PROGRAM MAIN
VAR		
	//INPUTS
	PrePump_Pressure_Int AT %I* : INT;
	Chamber_Penning_Int  AT %I* : INT;
	Chamber_Pirani_Int   AT %I* : INT;	
	GasLine_Pirani_Int   AT %I* : INT;
	Sample_BodyTemp      AT %I* : INT;					// Oven temperatures in 0.01 degC
	Sample_CapTemp       AT %I* : INT;
	Sample_TipTemp       AT %I* : INT;	
	Magnet_Temp          AT %I* : INT;
	
	Flow_Valve 			 AT %I* : INT;                  // Gas flow valve conductance 0-10 V
	
	TurboTOF_NO AT %I* : BOOL;	
	TurboTOF_ERR AT %I* : BOOL;
		
	
	// IMPORTANT! 
	// LEYBOLD AND BECKHOOF PLC USE DIFFERENT BYTE ORDER, be careful when linking to profibus
	// LEYBOLD:   0  1  2  3  4  5  6  7  8  9  10 11 12 13 14 15
	// BECKHOFF:  8  9  10 11 12 13 14 15 0  1  2  3  4  5  6  7 
	TurboMain_Overtemp AT %I* : BOOL;
	TurboMain_NO AT %I* : BOOL;
	TurboMain_ERR AT %I* : BOOL;
	TurboMain_Freq AT %I* : UINT;
	
	//OUTPUTS
	Penning_Enable AT %Q* : BOOL;
	LVPS_ON AT %Q* : BOOL;
	MPreVac_Valve AT %Q*: BOOL;
	TOFPreVac_Valve AT %Q* : BOOL;

	TurboTOF_enable AT %Q* : BOOL;
	TurboMain_enable AT %Q*: BOOL;
	TurboMain_Control AT %Q* : BOOL;

	Flow_Valve_Set AT %Q* : INT;    // Flow valve setpoint
	
	FlashInterlock AT %Q* : BOOL;	
	HVPS_ON AT %Q* : INT;
	Lamp1_Enable AT %Q* : BOOL;
	
	//ADS inputs: CONTROL PARAMETERS (PLC reads values and acts accordignly, ADS clients should set these values)
	GasLine_Enable :    BOOL := FALSE;
	Pumps_Enable :      BOOL := FALSE;      // Start pumping sequence
	PreVac_Valve_Lock : BOOL := FALSE;		// Ovverides auto valves and close prevac valves
	
	Sample_Flow_Set : REAL := 0;
	
	SampleX_MotionEnable : BOOL := FALSE;     // Motion enables and setpoints input
	SampleY_MotionEnable : BOOL := FALSE;  	
	SampleZ_MotionEnable : BOOL := FALSE;  	
	SampleX_MotionStop    : BOOL := FALSE;
	SampleY_MotionStop    : BOOL := FALSE;
	SampleZ_MotionStop    : BOOL := FALSE;
	
	FrameX_MotionEnable  : BOOL := FALSE;
	FrameY_MotionEnable  : BOOL := FALSE;
	FrameX_MotionStop     : BOOL := FALSE;
	FrameY_MotionStop     : BOOL := FALSE;
	
	MagnetY_MotionEnable : BOOL := FALSE;
	MagnetY_MotionStop    : BOOL := FALSE;
	
	SampleX_SetPoint : REAL := 0;
	SampleY_SetPoint : REAL := 0;
	SampleZ_SetPoint : REAL := 0;
	FrameX_SetPoint  : REAL := 0;
	FrameY_SetPoint  : REAL := 0;
	MagnetY_SetPoint  : REAL := 0;
	
	//ADS outputs: READ ONLY (PLC updates them at every cycle, ADS clients should just read)
	Chamber_Pressure : REAL;				// Main chamber pressure in mBars
	GasLine_Pressure : REAL;
	PreVac_Pressure  : REAL;                // PrePump line pressure
	PreVacValves_Open: BOOL;	            // Are valves open?

	Sample_Flow : REAL;
	
	TurboPump_ON: BOOL;
	TurboError: BOOL;	
	Turbo_NO:    BOOL;
	
	//Other vars
	PreVac_OK :  BOOL;						// Good prevacuum 
	MainVac_OK : BOOL;
	MainVac_TurboOK : BOOL;
	Oven_OverTEMP: BOOL;
	Pressure_Chamber_Manager: PressureChamber_MNG;
	
	//MOTION 
	manageAx_SampleX: manageAxis;
	manageAx_SampleY: manageAxis;
	manageAx_SampleZ: manageAxis;
	manageAx_FrameX: manageAxis;
	manageAx_FrameY: manageAxis;
	manageAx_MagnetY: manageAxis;	
		
	FrameX : AXIS_REF;
	FrameY : AXIS_REF;
	SampleZ : AXIS_REF;
	SampleX : AXIS_REF;
	SampleY : AXIS_REF;
	MagnetY : AXIS_REF;
	
	SampleX_Fw_End AT %I* : BOOL; // Limit switches
	SampleX_Bw_End AT %I* : BOOL;
	SampleY_Fw_End AT %I* : BOOL;
	SampleY_Bw_End AT %I* : BOOL; 
	SampleZ_Fw_End AT %I* : BOOL;
	SampleZ_Bw_End AT %I* : BOOL;  
	
	FrameX_Fw_End AT %I* : BOOL;
	FrameX_Bw_End AT %I* : BOOL; 
	FrameY_Fw_End AT %I* : BOOL;
	FrameY_Bw_End AT %I* : BOOL; 
	
	MagnetY_Fw_End AT %I* : BOOL;
	MagnetY_Bw_End AT %I* : BOOL;
END_VAR

//*** PROCESS INPUTS ***
//Get pressures in mbar (from ADC value)
Pressure_Chamber_Manager(penningInt := Chamber_Penning_Int, piraniInt := Chamber_Pirani_Int, penningOn => Penning_enable, pressureOut => Chamber_Pressure);
PreVac_Pressure := ConvertPressure_Pirani(PrePump_Pressure_Int);
GasLine_Pressure := ConvertPressure_Pirani(GasLine_Pirani_Int);

//*** MOTION ***
//Move axes
manageAx_SampleX(axis := SampleX, setPoint := SampleX_SetPoint, speed := PARAM.Sample_Movement_Speed, 
		 enable := SampleX_MotionEnable, stop:= SampleX_MotionStop, fwLimit := SampleX_Fw_End, bwLimit := SampleX_Bw_End);
		 
manageAx_SampleY(axis := SampleY, setPoint := SampleY_SetPoint, speed := PARAM.Sample_Movement_Speed, 
		 enable := SampleY_MotionEnable, stop:= SampleY_MotionStop, fwLimit := SampleY_Fw_End, bwLimit := SampleY_Bw_End);	 

manageAx_SampleZ(axis := SampleZ, setPoint := SampleZ_SetPoint, speed := PARAM.Sample_Movement_Speed, 
		 enable := SampleZ_MotionEnable, stop:= SampleZ_MotionStop, fwLimit := SampleZ_Fw_End, bwLimit := SampleZ_Bw_End);
		 
manageAx_FrameX(axis := FrameX,  setPoint := FrameX_SetPoint,  speed := PARAM.Frame_Movement_Speed , 
		 enable := FrameX_MotionEnable, stop:= FrameX_MotionStop, fwLimit := FrameX_Fw_End,  bwLimit := FrameX_Bw_End);

manageAx_FrameY(axis := FrameY,  setPoint := FrameY_SetPoint,  speed := PARAM.Frame_Movement_Speed , 
		 enable := FrameY_MotionEnable, stop:= FrameY_MotionStop, fwLimit := FrameY_Fw_End,  bwLimit := FrameY_Bw_End);
		 
manageAx_MagnetY(axis := MagnetY, setPoint := MagnetY_SetPoint, speed := PARAM.Sample_Movement_Speed, 
		 enable := MagnetY_MotionEnable, stop:= MagnetY_MotionStop, fwLimit := MagnetY_Fw_End, bwLimit := MagnetY_Bw_End);
		 
		 
//*** SAFETY CHECKS ***
// Compute status variables
Oven_OverTEMP   := Sample_BodyTemp > PARAM.Oven_MaxTemp OR Sample_TipTemp > PARAM.Oven_MaxTemp; // OR Sample_CapTemp > PARAM.Oven_MaxTemp Prevent overtemp of oven
TurboError 		:= TurboTOF_ERR AND TurboMain_ERR;
Turbo_NO        := TurboTOF_NO AND TurboMain_NO; 
MainVac_OK      := Chamber_Pressure > 0 AND Chamber_Pressure < PARAM.MainVac_Ok_Threshold; // Negative pressure means sensor error or sensor disconnected
MainVac_TurboOK := Chamber_Pressure > 0 AND Chamber_Pressure < PARAM.TurboStart_Threshold;
PreVac_OK       := PreVac_Pressure  > 0 AND PreVac_Pressure  < PARAM.PreVac_Ok_Threshold;


// Decide actions based on status
PreVacValves_Open := NOT PreVac_Valve_Lock AND ( PreVac_OK OR NOT MainVac_TurboOK );
TurboPump_ON := PreVac_Ok AND Pumps_Enable AND MainVac_TurboOK AND NOT TurboError;
LVPS_ON := MainVac_TurboOK AND NOT Oven_OverTEMP;

// Sample Valve
Sample_Flow := INT_TO_REAL(Flow_Valve) / 32767; // convert int to float in range 0-1
Sample_Flow_Set := MAX( MIN( Sample_Flow_Set, 1), 0);
Flow_Valve_Set := REAL_TO_INT( Sample_Flow_Set * 32767) * BOOL_TO_INT(MainVac_TurboOK) * BOOL_TO_INT(GasLine_Enable);  // If vented, valve is closed

// Actuate outputs (when one action controls more than one output)
MPreVac_Valve   := PreVacValves_Open;
TOFPreVac_Valve := PreVacValves_Open;
TurboTOF_enable  := TurboPump_ON;
TurboMain_enable := TurboPump_ON;
TurboMain_control := TRUE; // Tell pump that control is through Profibus and ignore other signals

IF MainVac_OK AND Turbo_NO THEN
	FlashInterlock := TRUE;
	HVPS_ON := PARAM.HVPS_SafetyLoop_Current;
ELSE
	FlashInterlock := FALSE;
	HVPS_ON := 0;
END_IF

END_PROGRAM

(* stored: Version 1.1.0.1, ProductVersion 3.1.4024.4
   POU MAIN: Id {bebe6b61-023e-4d51-b092-c239fd7bc0f8}, SpecialFunc None *)
